FUNCTION_BLOCK UNIT_Blikkenvullijn EXTENDS FB_Machine_PackML IMPLEMENTS  ITF_UNIT_Blikkenvullijn
VAR
	fb_mem									: STRUCT_UNIT_Blikkenvullijn;
	
	//Custom logic
	EM_Can_Supply 							: EM_Can_Supply;		//Replace with actual block not function
	//CM_TurningDevice						: CM_Motor;
	CM_Outfeed_ProductionLineSensor			: CM_Sensor;
	
	//PackML machine's
	EM_Filling								: FB_Machine_PackML;		//Replace with actual block not function
	EM_CheckWeigher							: FB_Machine_PackML;		//Replace with actual block not function
	EM_BottomSeal							: FB_Machine_PackML;		//Replace with actual block not function
	EM_Labeller								: FB_Machine_PackML;		//Replace with actual block not function
	EM_TurningDevice						: FB_Machine_PackML;		//Replace with actual block not function
	EM_StampUnit							: FB_Machine_PackML;		//Replace with actual block not function
	EM_SealShrink							: FB_Machine_PackML;		//Replace with actual block not function
	
	//Transport logic
	EM_Infeed_CheckWeigher					: EM_Transport;
	EM_Transport_Checkweigher_BottomSeal	: EM_Transport_Mechanische_Stop;
	EM_Transport_BottomSeal_Labeller		: EM_Transport_Mechanische_Stop;
	EM_Transport_TurningDevice_StampUnit	: EM_Transport;
	EM_Transport_StampUnit_SealShrink		: EM_Transport_Mechanische_Stop;
	
	//Management Logic
	AlarmHandler 							: AlarmHandler;
	ModeSelect								: ModeSelect;
END_VAR

(*
$$$$$$$$\                                                                   $$\       $$$$$$$$\                     $$\                                         $$\                     
$$  _____|                                                                  $$ |      $$  _____|                    \__|                                        \__|                    
$$ |   $$$$$$\   $$$$$$\  $$$$$$$\  $$\  $$\  $$\  $$$$$$\   $$$$$$\   $$$$$$$ |      $$ |      $$$$$$$\   $$$$$$\  $$\ $$$$$$$\   $$$$$$\   $$$$$$\   $$$$$$\  $$\ $$$$$$$\   $$$$$$\  
$$$$$\ \____$$\ $$  __$$\ $$  __$$\ $$ | $$ | $$ |$$  __$$\ $$  __$$\ $$  __$$ |      $$$$$\    $$  __$$\ $$  __$$\ $$ |$$  __$$\ $$  __$$\ $$  __$$\ $$  __$$\ $$ |$$  __$$\ $$  __$$\ 
$$  __|$$$$$$$ |$$ |  \__|$$ |  $$ |$$ | $$ | $$ |$$ /  $$ |$$ /  $$ |$$ /  $$ |      $$  __|   $$ |  $$ |$$ /  $$ |$$ |$$ |  $$ |$$$$$$$$ |$$$$$$$$ |$$ |  \__|$$ |$$ |  $$ |$$ /  $$ |
$$ |  $$  __$$ |$$ |      $$ |  $$ |$$ | $$ | $$ |$$ |  $$ |$$ |  $$ |$$ |  $$ |      $$ |      $$ |  $$ |$$ |  $$ |$$ |$$ |  $$ |$$   ____|$$   ____|$$ |      $$ |$$ |  $$ |$$ |  $$ |
$$ |  \$$$$$$$ |$$ |      $$ |  $$ |\$$$$$\$$$$  |\$$$$$$  |\$$$$$$  |\$$$$$$$ |      $$$$$$$$\ $$ |  $$ |\$$$$$$$ |$$ |$$ |  $$ |\$$$$$$$\ \$$$$$$$\ $$ |      $$ |$$ |  $$ |\$$$$$$$ |
\__|   \_______|\__|      \__|  \__| \_____\____/  \______/  \______/  \_______|      \________|\__|  \__| \____$$ |\__|\__|  \__| \_______| \_______|\__|      \__|\__|  \__| \____$$ |
                                                                                                          $$\   $$ |                                                          $$\   $$ |
                                                                                                          \$$$$$$  |                                                          \$$$$$$  |
                                                                                                           \______/                                                            \______/ 
*)
//********************************ZEROING***********************************

//Make PackML values FALSE						//MAKE SURE UNDERLYING BLOCKS GETS ZERO-ED TOO!
ZeroAllVar();
EM_Can_Supply.ZeroAllVar();
EM_Filling.ZeroAllVar();
EM_Infeed_CheckWeigher.ZeroAllVar();
EM_CheckWeigher.ZeroAllVar();
EM_Transport_Checkweigher_BottomSeal.ZeroAllVar();
EM_BottomSeal.ZeroAllVar();
EM_Transport_BottomSeal_Labeller.ZeroAllVar();
EM_Labeller.ZeroAllVar();
EM_TurningDevice.ZeroAllVar();
EM_Transport_TurningDevice_StampUnit.ZeroAllVar();
EM_StampUnit.ZeroAllVar();
EM_Transport_StampUnit_SealShrink.ZeroAllVar();
EM_SealShrink.ZeroAllVar();


//********************************Exeptionhandling***********************************
// Puts line in HOLDING if a module is SUSPENDING
IF 	EM_Can_Supply.State 							= E_State_PackML.HOLDING OR
		EM_Filling.State 							= E_State_PackML.HOLDING OR
		EM_Infeed_CheckWeigher.State				= E_State_PackML.HOLDING OR
		EM_CheckWeigher.State 						= E_State_PackML.HOLDING OR
		EM_Transport_Checkweigher_BottomSeal.State	= E_State_PackML.HOLDING OR
		EM_BottomSeal.State							= E_State_PackML.HOLDING OR
		EM_Transport_BottomSeal_Labeller.State		= E_State_PackML.HOLDING OR
		EM_Labeller.State 							= E_State_PackML.HOLDING OR
		EM_TurningDevice.State						= E_State_PackML.HOLDING OR
		EM_Transport_TurningDevice_StampUnit.State	= E_State_PackML.HOLDING OR
		EM_StampUnit.State							= E_State_PackML.HOLDING OR
		EM_Transport_StampUnit_SealShrink.State		= E_State_PackML.HOLDING OR
		EM_SealShrink.State 						= E_State_PackML.HOLDING THEN
	fbPackML_mem.Suspend := TRUE;
	EM_Can_Supply.Suspend();
	EM_Filling.Suspend();
	EM_Infeed_CheckWeigher.Stop();
	EM_CheckWeigher.Suspend();
	EM_Transport_Checkweigher_BottomSeal.Stop();
	EM_BottomSeal.Suspend();
	EM_Transport_BottomSeal_Labeller.Stop();
	EM_Labeller.Suspend();
	EM_TurningDevice.Suspend();
	EM_Transport_TurningDevice_StampUnit.Stop();
	EM_StampUnit.Suspend();
	EM_Transport_StampUnit_SealShrink.Stop();
	EM_SealShrink.Suspend();
END_IF

//Puts line in ABORT if told so
IF fb_mem.CS.Abort AND ModeSelect.Auto() OR fb_mem.HMI.Abort AND ModeSelect.Manueel() THEN
	fbPackML_mem.Abort 							:= TRUE;
	EM_Can_Supply.Abort();
	EM_Filling.Abort();
	EM_Infeed_CheckWeigher.Abort();
	EM_CheckWeigher.Abort();
	EM_Transport_Checkweigher_BottomSeal.Abort();
	EM_BottomSeal.Abort();
	EM_Transport_BottomSeal_Labeller.Abort();
	EM_Labeller.Abort();
	EM_TurningDevice.Abort();
	EM_Transport_TurningDevice_StampUnit.Abort();
	EM_StampUnit.Abort();
	EM_Transport_StampUnit_SealShrink.Abort();
	EM_SealShrink.Abort();
END_IF
// Puts line in STOPPING if told so
IF fb_mem.CS.Stop AND ModeSelect.Auto() OR fb_mem.HMI.Stop AND ModeSelect.Manueel() THEN
	fbPackML_mem.Stop							:= TRUE;
	EM_Can_Supply.Stop();
	EM_Filling.Stop();
	EM_Infeed_CheckWeigher.Stop();
	EM_CheckWeigher.Stop();
	EM_Transport_Checkweigher_BottomSeal.Stop();
	EM_BottomSeal.Stop();
	EM_Transport_BottomSeal_Labeller.Stop();
	EM_Labeller.Stop();
	EM_TurningDevice.Stop();
	EM_Transport_TurningDevice_StampUnit.Stop();
	EM_StampUnit.Stop();
	EM_Transport_StampUnit_SealShrink.Stop();
	EM_SealShrink.Stop();
END_IF



//********************************Action case***********************************
CASE fbPackML_mem.State OF
	E_State_PackML.IDLE 			: 
		IF fb_mem.CS.Start AND ModeSelect.Auto() OR fb_mem.HMI.Start AND ModeSelect.Manueel() THEN
			fbPackML_mem.Start := TRUE;
		END_IF
	E_State_PackML.STARTING 		:
		// YET TO BE PROGRAMMED
	E_State_PackML.EXECUTE 			: 
		//Do nothing
	E_State_PackML.COMPLETE 		:
		IF fb_mem.CS.Clear AND ModeSelect.Auto() OR fb_mem.HMI.Clear AND ModeSelect.Manueel() THEN
			fbPackML_mem.Completing_SC := TRUE;
		END_IF
	E_State_PackML.RESETTING 		:
		//Reset the UNIT by reinitializing it
		FB_init(0,0);
		//When all the underlying modules have resetted, the state is completed
		IF 	EM_Can_Supply.State 						= E_State_PackML.IDLE AND
			EM_Filling.State 							= E_State_PackML.IDLE AND
			EM_Infeed_CheckWeigher						= E_State_PackML.IDLE AND
			EM_CheckWeigher.State 						= E_State_PackML.IDLE AND
			EM_Transport_Checkweigher_BottomSeal.State	= E_State_PackML.IDLE AND
			EM_BottomSeal.State							= E_State_PackML.IDLE AND
			EM_Transport_BottomSeal_Labeller.State		= E_State_PackML.IDLE AND
			EM_Labeller.State 							= E_State_PackML.IDLE AND
			EM_TurningDevice.State						= E_State_PackML.IDLE AND
			EM_Transport_TurningDevice_StampUnit.State	= E_State_PackML.IDLE AND
			EM_StampUnit.State							= E_State_PackML.IDLE AND
			EM_Transport_StampUnit_SealShrink.State		= E_State_PackML.IDLE AND
			EM_SealShrink.State 						= E_State_PackML.IDLE THEN
		//State complete:
		fbPackML_mem.Resetting_SC := TRUE;
	END_IF
	E_State_PackML.HOLDING 			:
	E_State_PackML.HELD 			:
	E_State_PackML.UNHOLDING 		:
	E_State_PackML.SUSPENDING 		:
		IF (EM_Can_Supply.State 						= E_State_PackML.SUSPENDED OR
			EM_Can_Supply.State 						= E_State_PackML.HELD) AND
		   (EM_Filling.State 							= E_State_PackML.SUSPENDED OR
			EM_Filling.State 							= E_State_PackML.HELD) AND
		   (EM_Infeed_CheckWeigher						= E_State_PackML.SUSPENDED OR
			EM_Infeed_CheckWeigher						= E_State_PackML.HELD) AND
		   (EM_CheckWeigher.State 						= E_State_PackML.SUSPENDED OR
			EM_CheckWeigher.State 						= E_State_PackML.HELD) AND
		   (EM_Transport_Checkweigher_BottomSeal.State	= E_State_PackML.SUSPENDED OR
			EM_Transport_Checkweigher_BottomSeal.State	= E_State_PackML.HELD) AND
		   (EM_BottomSeal.State							= E_State_PackML.SUSPENDED OR
			EM_BottomSeal.State 						= E_State_PackML.HELD) AND
		   (EM_Transport_BottomSeal_Labeller.State		= E_State_PackML.SUSPENDED OR
			EM_Transport_BottomSeal_Labeller.State 		= E_State_PackML.HELD) AND
		   (EM_Labeller.State 							= E_State_PackML.SUSPENDED OR
			EM_Labeller.State 							= E_State_PackML.HELD) AND
		   (EM_TurningDevice.State						= E_State_PackML.SUSPENDED OR
			EM_TurningDevice.State 						= E_State_PackML.HELD) AND
		   (EM_Transport_TurningDevice_StampUnit.State	= E_State_PackML.SUSPENDED OR
			EM_Transport_TurningDevice_StampUnit.State	= E_State_PackML.HELD) AND
		   (EM_StampUnit.State							= E_State_PackML.SUSPENDED OR
			EM_StampUnit.State							= E_State_PackML.HELD) AND
		   (EM_Transport_StampUnit_SealShrink.State		= E_State_PackML.SUSPENDED OR
			EM_Transport_StampUnit_SealShrink.State		= E_State_PackML.HELD) AND
		   (EM_SealShrink.State 						= E_State_PackML.SUSPENDED OR 
			EM_SealShrink.State							= E_State_PackML.HELD) THEN
		fbPackML_mem.Suspending_SC := TRUE;
	END_IF
	
	E_State_PackML.SUSPENDED 		:
	IF 		EM_Can_Supply.State 						= E_State_PackML.UNHOLDING OR
			EM_Filling.State 							= E_State_PackML.UNHOLDING OR
			EM_Infeed_CheckWeigher						= E_State_PackML.UNHOLDING OR
			EM_CheckWeigher.State 						= E_State_PackML.UNHOLDING OR
			EM_Transport_Checkweigher_BottomSeal.State	= E_State_PackML.UNHOLDING OR
			EM_BottomSeal.State							= E_State_PackML.UNHOLDING OR
			EM_Transport_BottomSeal_Labeller.State		= E_State_PackML.UNHOLDING OR
			EM_Labeller.State 							= E_State_PackML.UNHOLDING OR
			EM_TurningDevice.State						= E_State_PackML.UNHOLDING OR
			EM_Transport_TurningDevice_StampUnit.State	= E_State_PackML.UNHOLDING OR
			EM_StampUnit.State							= E_State_PackML.UNHOLDING OR
			EM_Transport_StampUnit_SealShrink.State		= E_State_PackML.UNHOLDING OR
			EM_SealShrink.State 						= E_State_PackML.UNHOLDING THEN 
		fbPackML_mem.Unsuspend 							:= TRUE;
		EM_Can_Supply.Unsuspend();
		EM_Filling.Unsuspend();
		EM_Infeed_CheckWeigher.Start();
		EM_CheckWeigher.Unsuspend();
		EM_Transport_Checkweigher_BottomSeal.Start();
		EM_BottomSeal.Unsuspend();
		EM_Transport_BottomSeal_Labeller.Start();
		EM_Labeller.Unsuspend();
		EM_TurningDevice.Unsuspend();
		EM_Transport_TurningDevice_StampUnit.Start();
		EM_StampUnit.Unsuspend();
		EM_Transport_StampUnit_SealShrink.Start();
		EM_SealShrink.Unsuspend();
	END_IF
	E_State_PackML.UNSUSPENDING 	:
	E_State_PackML.ABORTED			:
		IF fb_mem.CS.Clear AND ModeSelect.Auto() OR fb_mem.HMI.Clear AND ModeSelect.Manueel() THEN
			fbPackML_mem.Clear 							:= TRUE;
			EM_Can_Supply.Clear();
			EM_Filling.Clear();
			EM_Infeed_CheckWeigher.Clear();
			EM_CheckWeigher.Clear();
			EM_Transport_Checkweigher_BottomSeal.Clear();
			EM_BottomSeal.Clear();
			EM_Transport_BottomSeal_Labeller.Clear();
			EM_Labeller.Clear();
			EM_TurningDevice.Clear();
			EM_Transport_TurningDevice_StampUnit.Clear();
			EM_StampUnit.Clear();
			EM_Transport_StampUnit_SealShrink.Clear();
			EM_SealShrink.Clear();
		END_IF
	E_State_PackML.ABORTING			:
		IF 	EM_Can_Supply.State 							= E_State_PackML.ABORTED OR
				EM_Filling.State 							= E_State_PackML.ABORTED OR
				EM_Infeed_CheckWeigher.State				= E_State_PackML.ABORTED OR
				EM_CheckWeigher.State 						= E_State_PackML.ABORTED OR
				EM_Transport_Checkweigher_BottomSeal.State	= E_State_PackML.ABORTED OR
				EM_BottomSeal.State							= E_State_PackML.ABORTED OR
				EM_Transport_BottomSeal_Labeller.State		= E_State_PackML.ABORTED OR
				EM_Labeller.State 							= E_State_PackML.ABORTED OR
				EM_TurningDevice.State						= E_State_PackML.ABORTED OR
				EM_Transport_TurningDevice_StampUnit.State	= E_State_PackML.ABORTED OR
				EM_StampUnit.State							= E_State_PackML.ABORTED OR
				EM_Transport_StampUnit_SealShrink.State		= E_State_PackML.ABORTED OR
				EM_SealShrink.State 						= E_State_PackML.ABORTED THEN
			fbpackML_mem.Aborting_SC := TRUE;
		END_IF
	E_State_PackML.CLEARING 		:
		IF 	EM_Can_Supply.State 							= E_State_PackML.STOPPED OR
				EM_Filling.State 							= E_State_PackML.STOPPED OR
				EM_Infeed_CheckWeigher.State				= E_State_PackML.STOPPED OR
				EM_CheckWeigher.State 						= E_State_PackML.STOPPED OR
				EM_Transport_Checkweigher_BottomSeal.State	= E_State_PackML.STOPPED OR
				EM_BottomSeal.State							= E_State_PackML.STOPPED OR
				EM_Transport_BottomSeal_Labeller.State		= E_State_PackML.STOPPED OR
				EM_Labeller.State 							= E_State_PackML.STOPPED OR
				EM_TurningDevice.State						= E_State_PackML.STOPPED OR
				EM_Transport_TurningDevice_StampUnit.State	= E_State_PackML.STOPPED OR
				EM_StampUnit.State							= E_State_PackML.STOPPED OR
				EM_Transport_StampUnit_SealShrink.State		= E_State_PackML.STOPPED OR
				EM_SealShrink.State 						= E_State_PackML.STOPPED THEN
			fbpackML_mem.Clearing_SC := TRUE;
		END_IF
	E_State_PackML.STOPPING 		:
	E_State_PackML.STOPPED 			:
		IF fb_mem.CS.Reset AND ModeSelect.Auto() OR fb_mem.HMI.Reset AND ModeSelect.Manueel() THEN
			fbPackML_mem.Reset 							:= TRUE;
			EM_Can_Supply.Reset();
			EM_Filling.Reset();
			EM_Infeed_CheckWeigher.Reset();
			EM_CheckWeigher.Reset();
			EM_Transport_Checkweigher_BottomSeal.Reset();
			EM_BottomSeal.Reset();
			EM_Transport_BottomSeal_Labeller.Reset();
			EM_Labeller.Reset();
			EM_TurningDevice.Reset();
			EM_Transport_TurningDevice_StampUnit.Reset();
			EM_StampUnit.Reset();
			EM_Transport_StampUnit_SealShrink.Reset();
			EM_SealShrink.Reset();
		END_IF 
END_CASE

METHOD FB_init : BOOL
VAR_INPUT
	bInitRetains : BOOL; // if TRUE, the retain variables are initialized (warm start / cold start)
	bInCopyCode : BOOL;  // if TRUE, the instance afterwards gets moved into the copy code (online change)
END_VAR
//**************************INITIATE**************************//
//Custom logic
EM_Can_Supply.FB_init(0,0);
EM_TurningDevice.FB_init(0,0);
CM_Outfeed_ProductionLineSensor.FB_init(0,0);
	
//PackML machine's
EM_Filling.FB_init(0,0);
EM_CheckWeigher.FB_init(0,0);
EM_BottomSeal.FB_init(0,0);
EM_Labeller.FB_init(0,0);
EM_TurningDevice.FB_init(0,0);
EM_StampUnit.FB_init(0,0);
EM_SealShrink.FB_init(0,0);
	
//Transport logic
EM_Infeed_CheckWeigher.FB_init(0,0);
EM_Transport_Checkweigher_BottomSeal.FB_init(0,0);
EM_Transport_BottomSeal_Labeller.FB_init(0,0);
EM_Transport_TurningDevice_StampUnit.FB_init(0,0);
EM_Transport_StampUnit_SealShrink.FB_init(0,0);
END_METHOD

END_FUNCTION_BLOCK

(* stored: Version 1.1.0.1, ProductVersion 3.1.4024.12
   POU UNIT_Blikkenvullijn: Id {2692377b-29af-456d-aace-ede4a94c185d}, SpecialFunc None
   Method FB_init: Id {e016cb9e-71c8-4e78-924d-1e46be021f7d} *)
